VISUALIZATION VISU_State_gray_red  // 12x17
VAR_IN_OUT
	state : BOOL;
END_VAR
    Ellipse (0,5 10x10), colour toggle: state
END_VISUALIZATION

(* stored: Version 1.1.0.1, ProductVersion 3.1.4018.5
   Visu VISU_State_gray_red: Id {c2c446bd-36eb-464e-8032-0176a2a85cc6} *)
